% RSLogix 500 project pressure_control.RSS, saved by version 8.30.00.16 %
PROJECT "UNTITLED"    % processor: Bul.1763 MicroLogix 1100 Series B %

PROGRAM FILES
  LAD 2   13 rungs

DATA FILES
  O0 OUTPUT  4 elements
  I1 INPUT  6 elements
  S2 STATUS  66 elements
  B3 BINARY  10 elements
  T4 TIMER  1 elements
  C5 COUNTER  1 elements
  R6 CONTROL  1 elements
  N7 INTEGER  16 elements
  F8 DUMYTARGET  1 elements
  F9 PARAMETERS  32 elements
  F10 PID_FLOATS  30 elements

LADDER 2
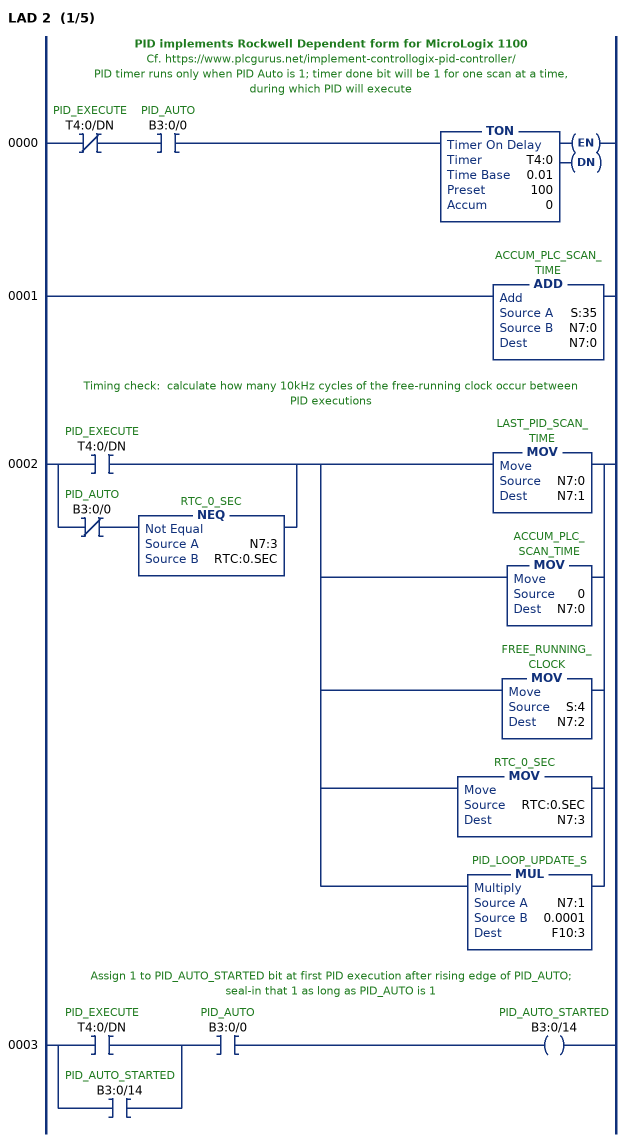
% Rung: 0 %
% TITLE: PID implements Rockwell Dependent form for MicroLogix 1100 %
% Cf. https://www.plcgurus.net/implement-controllogix-pid-controller/
% 
% PID timer runs only when PID Auto is 1; timer done bit will be 1 for one scan at a time, during which PID will execute %
SOR XIO T4:0/DN XIC B3:0/0 TON T4:0 0.01 100 0 EOR
%   T4:0/DN  PID_EXECUTE %
%   B3:0/0  PID_AUTO %
% Rung: 1 %
SOR ADD S:35 N7:0 N7:0 EOR
%   S:35  "Last 1 ms Scan Time" %
%   N7:0  ACCUM_PLC_SCAN_TIME %
% Rung: 2 %
% Timing check:  calculate how many 10kHz cycles of the free-running clock occur between PID executions %
SOR BST XIC T4:0/DN NXB XIO B3:0/0 NEQ N7:3 RTC:0.SEC BND BST MOV N7:0 N7:1 NXB MOV 0 N7:0 NXB MOV S:4 N7:2 NXB MOV RTC:0.SEC N7:3 NXB MUL N7:1 0.0001 F10:3 BND EOR
%   T4:0/DN  PID_EXECUTE %
%   B3:0/0  PID_AUTO %
%   N7:3  RTC_0_SEC %
%   N7:0  ACCUM_PLC_SCAN_TIME %
%   N7:1  LAST_PID_SCAN_TIME %
%   S:4  "Time Base" %
%   N7:2  FREE_RUNNING_CLOCK %
%   F10:3  PID_LOOP_UPDATE_S %
% Rung: 3 %
% Assign 1 to PID_AUTO_STARTED bit at first PID execution after rising edge of PID_AUTO; seal-in that 1 as long as PID_AUTO is 1 %
SOR BST XIC T4:0/DN NXB XIC B3:0/14 BND XIC B3:0/0 OTE B3:0/14 EOR
%   T4:0/DN  PID_EXECUTE %
%   B3:0/14  PID_AUTO_STARTED %
%   B3:0/0  PID_AUTO %

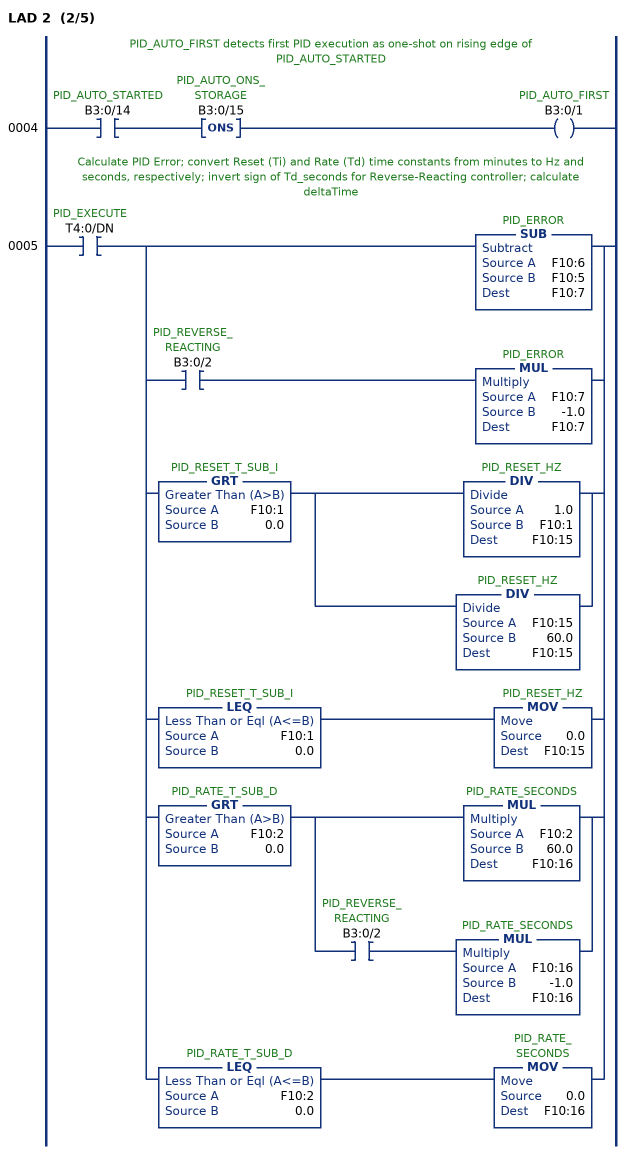
% Rung: 4 %
% PID_AUTO_FIRST detects first PID execution as one-shot on rising edge of PID_AUTO_STARTED %
SOR XIC B3:0/14 ONS B3:0/15 OTE B3:0/1 EOR
%   B3:0/14  PID_AUTO_STARTED %
%   B3:0/15  PID_AUTO_ONS_STORAGE %
%   B3:0/1  PID_AUTO_FIRST %
% Rung: 5 %
% Calculate PID Error; convert Reset (Ti) and Rate (Td) time constants from minutes to Hz and seconds, respectively; invert sign of Td_seconds for Reverse-Reacting controller; calculate deltaTime %
SOR XIC T4:0/DN BST SUB F10:6 F10:5 F10:7 NXB XIC B3:0/2 MUL F10:7 -1.0 F10:7 NXB GRT F10:1 0.0 BST DIV 1.0 F10:1 F10:15 NXB DIV F10:15 60.0 F10:15 BND NXB LEQ F10:1 0.0 MOV 0.0 F10:15 NXB GRT F10:2 0.0 BST MUL F10:2 60.0 F10:16 NXB XIC B3:0/2 MUL F10:16 -1.0 F10:16 BND NXB LEQ F10:2 0.0 MOV 0.0 F10:16 BND EOR
%   T4:0/DN  PID_EXECUTE %
%   F10:6  PID_PRESENT_VALUE %
%   F10:5  PID_SETPOINT %
%   F10:7  PID_ERROR %
%   B3:0/2  PID_REVERSE_REACTING %
%   F10:1  PID_RESET_T_SUB_I %
%   F10:15  PID_RESET_HZ %
%   F10:2  PID_RATE_T_SUB_D %
%   F10:16  PID_RATE_SECONDS %

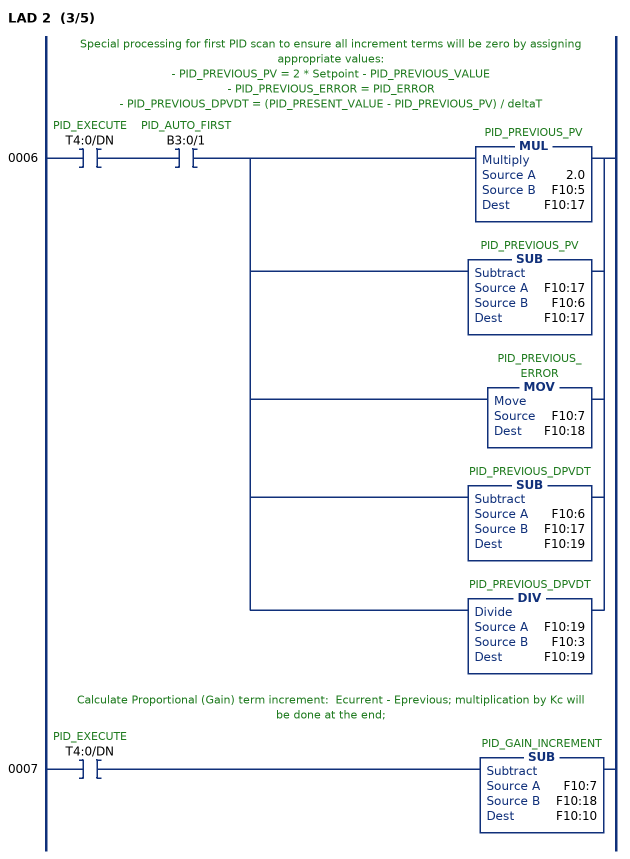
% Rung: 6 %
% Special processing for first PID scan to ensure all increment terms will be zero by assigning appropriate values:
% - PID_PREVIOUS_PV = 2 * Setpoint - PID_PREVIOUS_VALUE
% - PID_PREVIOUS_ERROR = PID_ERROR
% - PID_PREVIOUS_DPVDT = (PID_PRESENT_VALUE - PID_PREVIOUS_PV) / deltaT %
SOR XIC T4:0/DN XIC B3:0/1 BST BST MUL 2.0 F10:5 F10:17 NXB SUB F10:17 F10:6 F10:17 BND NXB MOV F10:7 F10:18 NXB BST SUB F10:6 F10:17 F10:19 NXB DIV F10:19 F10:3 F10:19 BND BND EOR
%   T4:0/DN  PID_EXECUTE %
%   B3:0/1  PID_AUTO_FIRST %
%   F10:5  PID_SETPOINT %
%   F10:17  PID_PREVIOUS_PV %
%   F10:6  PID_PRESENT_VALUE %
%   F10:7  PID_ERROR %
%   F10:18  PID_PREVIOUS_ERROR %
%   F10:19  PID_PREVIOUS_DPVDT %
%   F10:3  PID_LOOP_UPDATE_S %
% Rung: 7 %
% Calculate Proportional (Gain) term increment:  Ecurrent - Eprevious; multiplication by Kc will be done at the end; %
SOR XIC T4:0/DN SUB F10:7 F10:18 F10:10 EOR
%   T4:0/DN  PID_EXECUTE %
%   F10:7  PID_ERROR %
%   F10:18  PID_PREVIOUS_ERROR %
%   F10:10  PID_GAIN_INCREMENT %

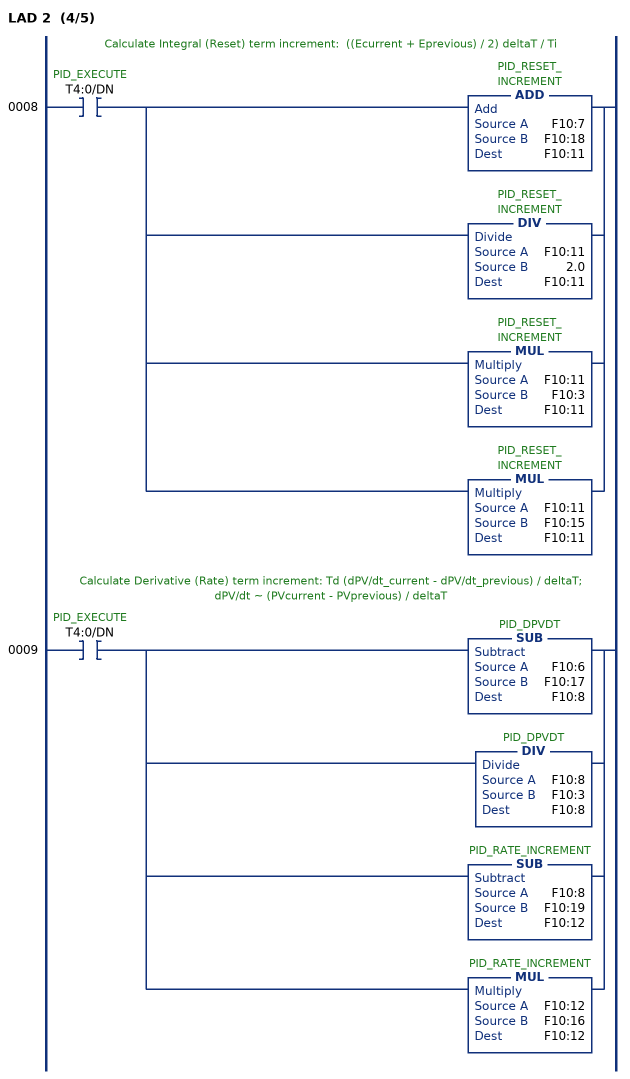
% Rung: 8 %
% Calculate Integral (Reset) term increment:  ((Ecurrent + Eprevious) / 2) deltaT / Ti %
SOR XIC T4:0/DN BST ADD F10:7 F10:18 F10:11 NXB DIV F10:11 2.0 F10:11 NXB MUL F10:11 F10:3 F10:11 NXB MUL F10:11 F10:15 F10:11 BND EOR
%   T4:0/DN  PID_EXECUTE %
%   F10:7  PID_ERROR %
%   F10:18  PID_PREVIOUS_ERROR %
%   F10:11  PID_RESET_INCREMENT %
%   F10:3  PID_LOOP_UPDATE_S %
%   F10:15  PID_RESET_HZ %
% Rung: 9 %
% Calculate Derivative (Rate) term increment: Td (dPV/dt_current - dPV/dt_previous) / deltaT; dPV/dt ~ (PVcurrent - PVprevious) / deltaT %
SOR XIC T4:0/DN BST SUB F10:6 F10:17 F10:8 NXB DIV F10:8 F10:3 F10:8 NXB SUB F10:8 F10:19 F10:12 NXB MUL F10:12 F10:16 F10:12 BND EOR
%   T4:0/DN  PID_EXECUTE %
%   F10:6  PID_PRESENT_VALUE %
%   F10:17  PID_PREVIOUS_PV %
%   F10:8  PID_DPVDT %
%   F10:3  PID_LOOP_UPDATE_S %
%   F10:19  PID_PREVIOUS_DPVDT %
%   F10:12  PID_RATE_INCREMENT %
%   F10:16  PID_RATE_SECONDS %

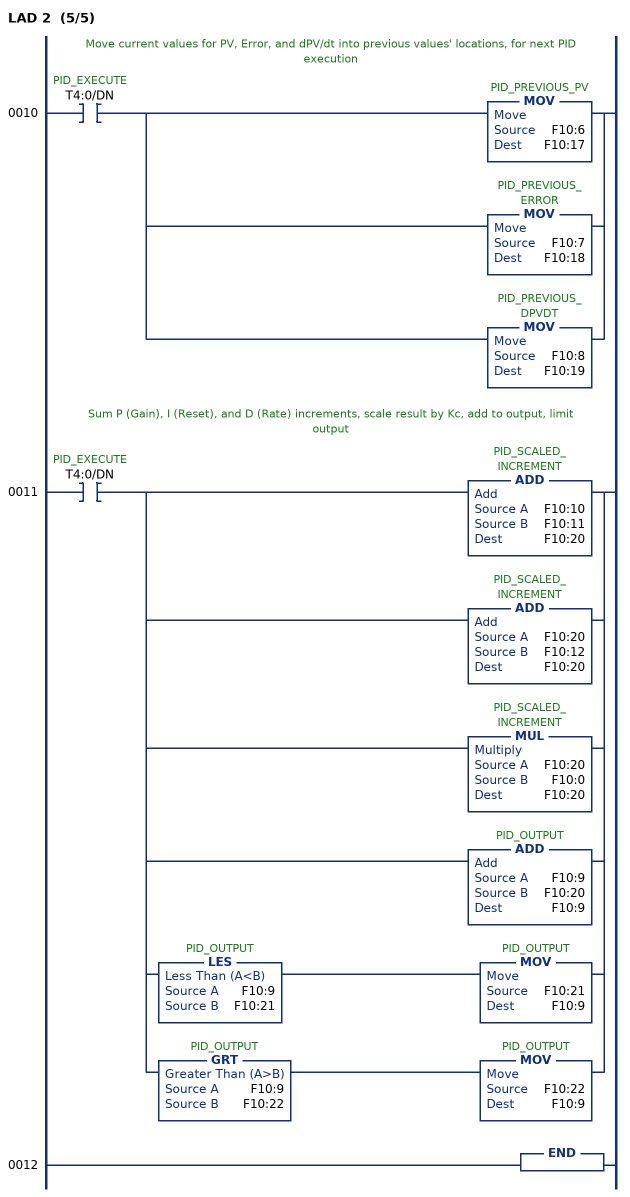
% Rung: 10 %
% Move current values for PV, Error, and dPV/dt into previous values' locations, for next PID execution %
SOR XIC T4:0/DN BST MOV F10:6 F10:17 NXB MOV F10:7 F10:18 NXB MOV F10:8 F10:19 BND EOR
%   T4:0/DN  PID_EXECUTE %
%   F10:6  PID_PRESENT_VALUE %
%   F10:17  PID_PREVIOUS_PV %
%   F10:7  PID_ERROR %
%   F10:18  PID_PREVIOUS_ERROR %
%   F10:8  PID_DPVDT %
%   F10:19  PID_PREVIOUS_DPVDT %
% Rung: 11 %
% Sum P (Gain), I (Reset), and D (Rate) increments, scale result by Kc, add to output, limit output %
SOR XIC T4:0/DN BST ADD F10:10 F10:11 F10:20 NXB ADD F10:20 F10:12 F10:20 NXB MUL F10:20 F10:0 F10:20 NXB ADD F10:9 F10:20 F10:9 NXB LES F10:9 F10:21 MOV F10:21 F10:9 NXB GRT F10:9 F10:22 MOV F10:22 F10:9 BND EOR
%   T4:0/DN  PID_EXECUTE %
%   F10:10  PID_GAIN_INCREMENT %
%   F10:11  PID_RESET_INCREMENT %
%   F10:20  PID_SCALED_INCREMENT %
%   F10:12  PID_RATE_INCREMENT %
%   F10:0  PID_GAIN_K_SUB_C %
%   F10:9  PID_OUTPUT %
%   F10:21  PID_OUT_LOW_LIMIT %
%   F10:22  PID_OUT_HIGH_LIMIT %
% Rung: 12 %
SOR END EOR

OTHER DOCUMENTED ADDRESSES
  B3:0  PID_BITS
  F8:0  UNUSED_DUMMY_TARGET  "AdvancedHMIControls push values here to update Analog Value Displays"
  F9:0  PSIG
  F9:1  DELTA_PSIG_FROM_MODE
  F9:2  SPEED_0_100
  F9:3  RAMP_DELTA_SPEED
  PID_LAST_PV  
  PID_PREVIIOUS_PV  
  PID_REVERSE  

DATA TABLE (non-zero values as saved)
DATA B3
% B3:0 % 0X0004 0X0000 0X0000 0X0000 0X0000 0X0000 0X0000 0X0000 0X0000 0X0000
DATA T4
% .PRE .ACC %
% T4:0 % 100 0
DATA F10
% F10:5 % 0 0 0 0 50
% F10:20 % 0 0 100 0 0
